(* PLC project Unnamed, Unknown Unnamed 1 *)
(* stored: creationDateTime 2020-09-15T09:29:34, modificationDateTime 2023-06-14T00:00:00 *)

PROGRAM ElevatorControl
  VAR
    System_On AT %IX1.0 : BOOL;
    Floor1_Call AT %IX1.1 : BOOL;
    Floor2_Call AT %IX1.2 : BOOL;
    Floor1_Limit_Switch AT %IX1.3 : BOOL;
    Floor2_Limit_Switch AT %IX1.4 : BOOL;
    Floor1_Open_Door_Motor AT %QX1.0 : BOOL;
    Floor2_Open_Door_Motor AT %QX1.1 : BOOL;
    Floor1_Close_Door_Motor AT %QX1.2 : BOOL;
    Floor2_Close_Door_Motor AT %QX1.3 : BOOL;
    Floor1_Open_Door_Limit_Switch AT %IX1.5 : BOOL;
    Floor2_Open_Door_Limit_Switch AT %IX1.6 : BOOL;
    Floor1_Close_Door_Limit_Switch AT %IX1.7 : BOOL;
    Floor2_Close_Door_Limit_Switch AT %IX1.8 : BOOL;
    Pulley_Motor_Up AT %QX1.4 : BOOL;
    Pulley_Motor_Down AT %QX1.5 : BOOL;
    Door_Timer AT %TM1 : TON;
    Sequencer AT %IW1.0 : INT;
  END_VAR

            ElevatorControl
            
              
                System_On
              
              
                
                  Sequencer
                  1
                
              
            
            
              
                Sequencer
                
                  1
                
              
              
                
                  
                    
                      
                        Floor2_Call
                      
                      
                        
                          Floor2_Limit_Switch
                        
                      
                    
                  
                  
                    
                      Pulley_Motor_Up
                      true
                    
                    
                      Sequencer
                      2
                    
                  
                  
                    
                      
                        
                          Floor1_Call
                        
                        
                          
                            Floor1_Limit_Switch
                          
                        
                      
                    
                    
                      
                        Pulley_Motor_Down
                        true
                      
                      
                        Sequencer
                        3
                      
                    
                  
                
              
            
            
              
                Sequencer
                
                  2
                
              
              
                
                  
                    Floor2_Limit_Switch
                  
                  
                    
                      Pulley_Motor_Up
                      false
                    
                    
                      Floor2_Open_Door_Motor
                      true
                    
                    
                      
                        Floor2_Open_Door_Limit_Switch
                      
                      
                        
                          Floor2_Open_Door_Motor
                          false
                        
                        
                          TON
                          Door_Timer
                          
                            
                              
                            
                            true
                          
                        
                        
                          Sequencer
                          4
                        
                      
                    
                  
                
              
            
            
              
                Sequencer
                
                  3
                
              
              
                
                  
                    Floor1_Limit_Switch
                  
                  
                    
                      Pulley_Motor_Down
                      false
                    
                    
                      Floor1_Open_Door_Motor
                      true
                    
                    
                      
                        Floor1_Open_Door_Limit_Switch
                      
                      
                        
                          Floor1_Open_Door_Motor
                          false
                        
                        
                          TON
                          Door_Timer
                          
                            
                              
                            
                            true
                          
                        
                        
                          Sequencer
                          5
                        
                      
                    
                  
                
              
            
            
              
                Sequencer
                
                  4
                
              
              
                
                  
                    Door_Timer.Q
                  
                  
                    
                      Floor2_Close_Door_Motor
                      true
                    
                    
                      
                        Floor2_Close_Door_Limit_Switch
                      
                      
                        
                          Floor2_Close_Door_Motor
                          false
                        
                        
                          TON
                          Door_Timer
                          
                            
                              
                            
                            false
                          
                        
                        
                          Sequencer
                          1
                        
                      
                    
                  
                
              
            
            
              
                Sequencer
                
                  5
                
              
              
                
                  
                    Door_Timer.Q
                  
                  
                    
                      Floor1_Close_Door_Motor
                      true
                    
                    
                      
                        Floor1_Close_Door_Limit_Switch
                      
                      
                        
                          Floor1_Close_Door_Motor
                          false
                        
                        
                          TON
                          Door_Timer
                          
                            
                              
                            
                            false
                          
                        
                        
                          Sequencer
                          1
                        
                      
                    
                  
                
              
            
          
END_PROGRAM

CONFIGURATION Config0
  RESOURCE Res0 ON PLC
    TASK task0(INTERVAL := T#20ms, PRIORITY := 0);
    PROGRAM instance0 WITH task0 : ElevatorControl;
  END_RESOURCE
END_CONFIGURATION
